{attribute 'linkalways'} 
{attribute 'no_explicit_call' := 'This FB is a CLASS and must be accessed using methods or properties'}
{attribute 'enable_dynamic_creation'}
FUNCTION_BLOCK Node_F_VN_FillContainerExp_TcVnKeyPoint EXTENDS VisionNode
VAR
    ipContainer : _ITcVnContainer;
    stValue : _TcVnKeyPoint;
    nStartIdx : _ULINT(0);
    nCount : _ULINT(0);
    hrPrev : _HRESULT(S_OK);
    hresult : _HRESULT(S_OK);
END_VAR

METHOD PUBLIC  Clone : I_Node
VAR
    pNode : POINTER TO Node_F_VN_FillContainerExp_TcVnKeyPoint;
END_VAR
pNode := __NEW(Node_F_VN_FillContainerExp_TcVnKeyPoint);
Clone := pNode^;
END_METHOD

METHOD FB_init : BOOL
VAR_INPUT
    bInitRetains : BOOL; // if TRUE, the retain variables are initialized (warm start / cold start)
    bInCopyCode : BOOL;  // if TRUE, the instance afterwards gets moved into the copy code (online change)
END_VAR
AddInput('ipContainer', ipContainer);
AddInput('stValue', stValue);
AddParameter('nStartIdx', nStartIdx);
AddParameter('nCount', nCount);
AddInput('hrPrev', hrPrev);
AddOutput('ipContainer', ipContainer);
AddOutput('hresult',hresult);
END_METHOD

METHOD PROTECTED OnExecute
hresult.Value := F_VN_FillContainerExp_TcVnKeyPoint(
    ipContainer := ipContainer.Value,
    stValue := stValue.Value,
    nStartIdx := nStartIdx.Value,
    nCount := nCount.Value,
    hrPrev:= hrPrev.Value);
END_METHOD

METHOD PUBLIC PreExecutionCheck
VAR_INPUT
    Check : I_PreExecutionChecks;
END_VAR
Check.IsTrue(ipContainer.IsValid, 'ipContainer must be a valid container');
Check.IsTrue(ipContainer.IsType(TC_GLOBAL_CONST_LIST.ContainerType_Vector_TcVnKeyPoint), 'ipContainer contains incorrect type');
END_METHOD

END_FUNCTION_BLOCK

(* stored: Version 1.1.0.1, ProductVersion 3.1.4026.13
   POU Node_F_VN_FillContainerExp_TcVnKeyPoint: Id {109b555f-aa17-466b-aa3f-4ef4f2b67f57}, SpecialFunc None
   Folder Constructor: Id {e52a9461-16f0-4444-8e14-6eb2ce751ff4}
   Method Clone: Id {7cc36891-daaf-41eb-8346-2669be1064bf}
   Method FB_init: Id {d445001e-ee6d-4677-beb6-2fbcb0c0f12a}
   Method OnExecute: Id {6c420f5c-4740-4aef-82e1-3e6b5a8bc6dc}
   Method PreExecutionCheck: Id {0ed13564-c3b6-4cc8-94e5-604f9aa105e1} *)
